(* LS Electric XG5000 project: ADC_EIP_StatusFB *)
(* This project is for getting the EtherNet/IP General and Extended Status from XBL-EIPT Module *)
(* PLC LSPLC *)
(* module base 0 slot 0: Input/Output Module:XEM-DN/DP32HP (DC 24V Input, Transistor Output, 32 Contacts) *)
(* module base 0 slot 1: Internal Positioning:XBF-PO06E (Open Collector Type, 6 Axis) *)
(* module base 0 slot 2: EtherNet/IP:XBL-EIPT (EtherNet/IP communication module, electrical) *)
VAR_GLOBAL
    in1 : ARRAY[0..249] OF BYTE;
    out1 : ARRAY[0..249] OF BYTE;
END_VAR

FUNCTION_BLOCK EIP_Get_Status
(* This function block can be used to get the general and extended status information for a EIP P2P index *)
VAR_INPUT
    Execute : BOOL; (* Execute function block on rising edge. *)
    EIPT_Slot_Number : USINT; (* Slot number of the XBL-EIPT module. Valid values are 2~7. *)
    P2P_Index_Number : USINT; (* P2P index number that the status should be fetched for. Valid Values are 0-31 *)
END_VAR
VAR_OUTPUT
    Done : BOOL; (* Status that function block has completed *)
    Status : SINT; (* Status of the function block.  -1 means an invalid EIPT_Slot_Number was entered. / -2 means an invalid P2P_Index_Number was entered. / 0 and positive values are CP_MSG status values. *)
    General_Status_Data : USINT; (* 1 Byte of General Status information *)
    Extended_Status_Data00 : UINT; (* 1st word of Extend Status data *)
    Extended_Status_Data01 : UINT; (* 2nd word of Extend Status data *)
    Extended_Status_Data02 : UINT; (* 3rd word of Extend Status data *)
    Extended_Status_Data03 : UINT; (* 4th word of Extend Status data *)
    Extended_Status_Data04 : UINT; (* 5th word of Extend Status data *)
    Extended_Status_Data05 : UINT; (* 6th word of Extend Status data *)
    Extended_Status_Data06 : UINT; (* 7th word of Extend Status data *)
    Extended_Status_Data07 : UINT; (* 8th word of Extend Status data *)
END_VAR
VAR
    CP_MSG_Instance : CP_MSG; (* message function block for retrieving status information.  Internal fb variable. *)
    Extended_Data_Size : USINT; (* number of words for extended status *)
    FrameCommand : WORD := 16#0111; (* frame command value for the CP_MSG function block *)
    REQ : BOOL; (* Internal REQ variable for CP_MSG function block. *)
    REQ_DATA : ARRAY[0..1499] OF BYTE; (* Data received from CP_MSG. Internal fb variable. *)
    REQ_SIZE : UINT; (* Request size for CP_MSG. Internal fb variable. *)
    RES_DATA : ARRAY[0..1499] OF BYTE; (* Result data of the CP_MSG.  Internal fb variable. *)
    tempDWORD : DWORD; (* temporary DWORD variable *)
    tempWORD1 : WORD; (* temporary WORD variable *)
    tempWORD2 : WORD; (* temporary WORD variable *)
END_VAR
(* 
AutomationDirect.com has provided this code for convenience. This sample code is provided "as-is" with no expressed or implied warranty. 
 If the end user includes any of the sample code (in whole or part), it is the user's responsibility to completely modify, integrate, and test any code to ensure it meets all system and 
 safety requirements for the intended application or system.
 *)

//Run CP_MSG to retrieve General Status and Extended Status while execute is true
IF (Execute)  THEN
		
	//Check for valid EIPT Slot number
	IF (EIPT_Slot_Number > 7) OR (EIPT_Slot_Number < 2) THEN
		Status := -1;
		
	//Check to make sure P2P Index number isn't higher then 31 since it shouldn't be	
	ELSIF (P2P_Index_Number > 31) THEN
		Status := -2;
	
	 ELSE		
		//Set REQ for CP_MSG to TRUE
		REQ := TRUE;
		
		// CP_MSG Frame Command must be 0x0111
		FrameCommand := 16#0111;
		WORD_BYTE(IN:=FrameCommand, LOW=>REQ_DATA[0], HIGH=>REQ_DATA[1]);
		
		//Object Count will be 16#01
 		REQ_DATA[4] := 16#01;
 		
 		//Data Type (5) and Object ID (7) has DWORD value of 16#00050007.  Data type conversions are used to make sure values are correctly translated to BYTE
 		tempDWORD := 16#00050007;
 		DWORD_WORD(IN:=tempDWORD, LOW=>tempWORD1, HIGH=>tempWORD2);
 		WORD_BYTE(IN:=tempWORD1, LOW=>REQ_DATA[8], HIGH=>REQ_DATA[9]);
 		WORD_BYTE(IN:=tempWORD2, LOW=>REQ_DATA[10], HIGH=>REQ_DATA[11]);
			 	
		// The offset of CP_MSG REQ_DATA is the P2P Block Number (0~31).  
		REQ_DATA[12] := USINT_TO_BYTE(IN:=P2P_Index_Number);
		
		//Length of the Data = 36.  General Status (2 BYTEs)+Extended Status Size (2 BYTEs) + Extended Status (32 BYTEs)
		REQ_DATA[16] :=  16#24;	 	
		
		//Set REQ_SIZE
		REQ_SIZE :=  16#14;
		
		//Copy general status and extended status information to function block outputs
		IF (CP_MSG_Instance.DONE) THEN
			General_Status_Data :=  BYTE_TO_USINT(RES_DATA[20]);
			
			Extended_Data_Size := BYTE_TO_USINT(RES_DATA[22]);
			
			IF (Extended_Data_Size >= 1) THEN
				tempWORD1 := BYTE_WORD(LOW:=RES_DATA[24], HIGH:=RES_DATA[25]);
				Extended_Status_Data00 := WORD_TO_UINT(tempWORD1);
			ELSE
				Extended_Status_Data00 := 0;
			END_IF;		
			
			IF (Extended_Data_Size >= 2) THEN
				tempWORD1 := BYTE_WORD(LOW:=RES_DATA[26], HIGH:=RES_DATA[27]);
				Extended_Status_Data01 := WORD_TO_UINT(tempWORD1);
			ELSE
				Extended_Status_Data01 := 0;
			END_IF;
				
			IF (Extended_Data_Size >= 3) THEN
				tempWORD1 := BYTE_WORD(LOW:=RES_DATA[28], HIGH:=RES_DATA[29]);
				Extended_Status_Data02 := WORD_TO_UINT(tempWORD1);
			ELSE	
				Extended_Status_Data02 := 0;
			END_IF;		
			
			IF (Extended_Data_Size >= 4) THEN
				tempWORD1 := BYTE_WORD(LOW:=RES_DATA[30], HIGH:=RES_DATA[31]);
				Extended_Status_Data03 := WORD_TO_UINT(tempWORD1);
			ELSE
				Extended_Status_Data03 := 0;
			END_IF;
				
			IF (Extended_Data_Size >= 5) THEN
				tempWORD1 := BYTE_WORD(LOW:=RES_DATA[32], HIGH:=RES_DATA[33]);
				Extended_Status_Data04 := WORD_TO_UINT(tempWORD1);
			ELSE
				Extended_Status_Data04 := 0;
			END_IF;		
			
			IF (Extended_Data_Size >= 6) THEN
				tempWORD1 := BYTE_WORD(LOW:=RES_DATA[34], HIGH:=RES_DATA[35]);
				Extended_Status_Data05 := WORD_TO_UINT(tempWORD1);
			ELSE
				Extended_Status_Data05 := 0;	
			END_IF;
				
			IF (Extended_Data_Size >= 7) THEN
				tempWORD1 := BYTE_WORD(LOW:=RES_DATA[36], HIGH:=RES_DATA[37]);
				Extended_Status_Data06 := WORD_TO_UINT(tempWORD1);
			ELSE
				Extended_Status_Data06 := 0;
			END_IF;
					
			IF (Extended_Data_Size >= 8) THEN
				tempWORD1 := BYTE_WORD(LOW:=RES_DATA[38], HIGH:=RES_DATA[39]);
				Extended_Status_Data07 := WORD_TO_UINT(tempWORD1);
			ELSE
				Extended_Status_Data07 := 0;
			END_IF;	
			
			
		END_IF;


		//copy CP_MSG status to this function blocks status
		Status := UINT_TO_SINT(CP_MSG_Instance.STAT);
		Done := CP_MSG_Instance.DONE;

	END_IF; // end check valid slot number and p2p index

// Actions for when execute is false.  
ELSE
	REQ := FALSE;
	Done := FALSE;
	Status := 0;
END_IF;
	
	
CP_MSG_Instance(REQ:=REQ, BASE:=0, SLOT:=EIPT_Slot_Number, REQ_DATA:=REQ_DATA, REQ_SIZE:=REQ_SIZE, TIMEOUT:=1000, RES_DATA:=RES_DATA);
END_FUNCTION_BLOCK

PROGRAM LD_Example (* task: Scan Program *)
VAR
    Execute_FB : BOOL;
    Extended_Status_Data00 : UINT;
    Extended_Status_Data01 : UINT;
    Extended_Status_Data02 : UINT;
    Extended_Status_Data03 : UINT;
    Extended_Status_Data04 : UINT;
    Extended_Status_Data05 : UINT;
    Extended_Status_Data06 : UINT;
    Extended_Status_Data07 : UINT;
    FB_Status : SINT; (* status of EIP_Get_Status FB *)
    General_Status_Data : USINT;
    Status_FB_Inst : EIP_Get_Status;
END_VAR

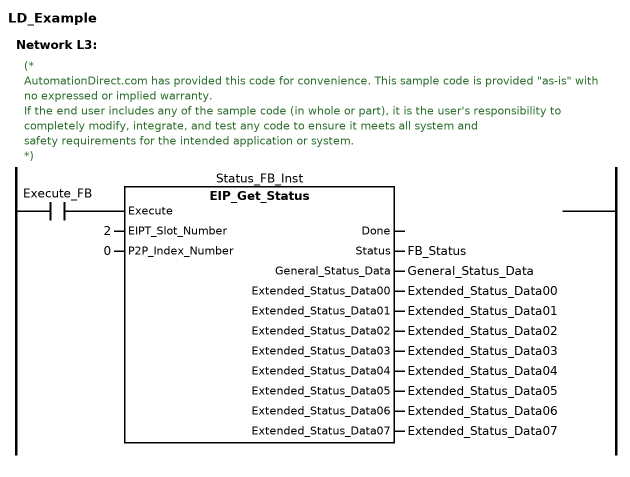
(* ( * / AutomationDirect.com has provided this code for convenience. This sample code is provided "as-is" with no expressed or implied warranty. / If the end user includes any of the sample code (in whole or part), it is the user's responsibility to completely modify, integrate, and test any code to ensure it meets all system and / safety requirements for the intended application or system. / * ) *)
(* Rung L3 *)
Status_FB_Inst(Execute := Execute_FB, EIPT_Slot_Number := 2, P2P_Index_Number := 0, Status => FB_Status, General_Status_Data => General_Status_Data, Extended_Status_Data00 => Extended_Status_Data00, Extended_Status_Data01 => Extended_Status_Data01, Extended_Status_Data02 => Extended_Status_Data02, Extended_Status_Data03 => Extended_Status_Data03, Extended_Status_Data04 => Extended_Status_Data04, Extended_Status_Data05 => Extended_Status_Data05, Extended_Status_Data06 => Extended_Status_Data06, Extended_Status_Data07 => Extended_Status_Data07);
END_PROGRAM

PROGRAM ST_Example (* task: Scan Program *)
(* this is a structured text example of the EIP_Get_Status function block. *)
VAR
    Execute_FB : BOOL; (* execute the function block *)
    INST_EIP_Get_Status : EIP_Get_Status; (* function block for getting EtherNet/IP general and extended status *)
END_VAR
(* 
AutomationDirect.com has provided this code for convenience. This sample code is provided "as-is" with no expressed or implied warranty. 
 If the end user includes any of the sample code (in whole or part), it is the user's responsibility to completely modify, integrate, and test any code to ensure it meets all system and 
 safety requirements for the intended application or system.
 *)
 
 
 INST_EIP_Get_Status(Execute:=Execute_FB, EIPT_Slot_Number:=2, P2P_Index_Number:=0);
END_PROGRAM